PROGRAM MAIN
VAR
END_VAR

END_PROGRAM

(* stored: Version 1.1.0.1
   POU MAIN: Id {8a349cbb-9d1a-4520-af1f-0a99ed2c2ee3} *)
